PROGRAM SingleCarrierMode
VAR
	(*key Command*)
	btn_Power:BOOL;
	btn_PowerOn: BOOL;
	btn_PowerOff: BOOL;
	TopPositionNew:LREAL:=100;
	TopVelocityNew:LREAL:=1;
	btn_TopMove:BOOL;
	btn_TopStop:BOOL;
	BottomPositionNew:LREAL:=100;
	BottomVelocityNew:LREAL:=1;
	btn_BottomMove:BOOL;
	btn_BottomStop:BOOL;
	(*Var*)
	fb_ton1:TON;
	fb_ton2:TON;
	fb_ton3:TON;
	(*Status*)
	State:DINT;
	Busy:BOOL;
	TopBusy:BOOL;
	BottomBusy:BOOL;
	InitDone:BOOL;
	tm_state: DINT;
	ts_state: DINT;
	bm_state: DINT;
	bs_state: DINT;
	(*PowerOff*)
	d_state: DINT;
	(*¼ì²âµ½ÏÞÎ»£¬»Ö¸´Move×´Ì¬*)
	FTrig_ReachLS: F_TRIG;
	FTrig_btn_GapMove: F_TRIG;
END_VAR

TopPositionActual:=(Pos_LeftTopLin+Pos_RightTopLin)/2;
TopVelocityActual:=(Velo_LeftTopLin+Velo_RightTopLin)/2;
BottomPositionActual:=(Pos_LeftBottomLin+Pos_RightBOttomLin)/2;
BottomVelocityActual:=(Velo_LeftBottomLin+Velo_RightBOttomLin)/2;
(*********************************************************************btn_PowerOn************************************************************)
IF btn_Power AND st_Power=0 THEN
	btn_PowerOn:=TRUE;
	btn_Power:=FALSE;
END_IF
IF btn_Power AND st_Power=1 THEN
	btn_PowerOff:=TRUE;
	btn_Power:=FALSE;
END_IF
(*********************************************************************btn_PowerOn************************************************************)

IF btn_PowerOn THEN
	A_CoupleAxisAndPowerOn();
END_IF
(******************************************************ÉÏµç×´Ì¬£¬²»´¦ÓÚñîºÏ×´Ì¬£¬ESTOP***********************************************)
IF NOT btn_PowerOff THEN
	IF st_Power=1 AND st_Couple<>1THEN
		Error:=TRUE;
		ErrorID:=101;
		FB_PlcEmergencyStop();
		LED_Error:=TRUE;
	END_IF
END_IF
(*********************************************************************Monitor All Carrirt Position***********************************************)
A_MonitoringAllAxis();
(*********************************************************************A_PosDiffDetection***********************************************)
A_PosDiffDetection();
(*********************************************************************btn_TopMove*****************************************************************)
IF InitDone THEN
	IF btn_TopMove AND NOT bottomBusy THEN
		TopBusy:=TRUE;
		btn_BottomMove:=FALSE;
		CASE tm_state OF
			0:
				FB_Move.Mode:=2;						(*1£ºgapÄ£Ê½£»2£ºµ¥ÁºÄ£Ê½£¬3£ºtaperÄ£Ê½*)
				FB_Move.CoupleState:=st_Couple;			(*ñîºÏ×´Ì¬ÊäÈë*)
				FB_Move.PowerState:=st_Power;			(*µçÔ´×´Ì¬ÊäÈë*)
				FB_Move.TopMove:=TRUE;				(*Execute TRUE*)
				FB_Move.TopPosition:=TopPositionNew;		(*Î»ÖÃ*)
				FB_Move.TopVelocity:=TopVelocityNew;		(*ËÙ¶È*)
				FB_Move();								(*Æô¶¯FB*)
				IF TopPositionNew-TopPositionActual>0.001 THEN	(*ÔË¶¯·½ÏòÖ¸Ê¾*)
					TopMoveIndicator:=1;
				ELSIF TopPositionNew-TopPositionActual<0.001 THEN
					TopMoveIndicator:=-1;
				ELSE
					TopMoveIndicator:=0;
				END_IF
				tm_state:=1;
			1:
				FB_Move();
				LED_Run:=TRUE;
				IF NOT FB_Move.TopDone THEN			(*ÔË¶¯Î´Íê³É£¬Ñ­»·*)
					tm_state:=1;
				ELSE									(*ÔË¶¯Íê³É£¬ÏÂÒ»²½*)
					tm_state:=88;
				END_IF
			88:
				btn_TopMove:=FALSE;					(*×´Ì¬»Ö¸´*)
				LED_Run:=FALSE;
				tm_state:=0;
				TopBusy:=FALSE;
		END_CASE
	END_IF
END_IF

(*********************************************************************btn_BottomMove*****************************************************************)
IF InitDone THEN
	IF btn_BottomMove AND NOT TopBusy THEN
		btn_TopMove:=FALSE;
		BottomBusy:=TRUE;
		CASE bm_state OF
			0:
				FB_Move.Mode:=2;						(*1£ºgapÄ£Ê½£»2£ºµ¥ÁºÄ£Ê½£¬3£ºtaperÄ£Ê½*)
				FB_Move.CoupleState:=st_Couple;			(*ñîºÏ×´Ì¬ÊäÈë*)
				FB_Move.PowerState:=st_Power;			(*µçÔ´×´Ì¬ÊäÈë*)
				FB_Move.BottomMove:=TRUE;				(*Execute TRUE*)
				FB_Move.BottomPosition:=BottomPositionNew;		(*Î»ÖÃ*)
				FB_Move.BottomVelocity:=BottomVelocityNew;		(*ËÙ¶È*)
				FB_Move();								(*Æô¶¯FB*)
				IF BottomPositionNew-BottomPositionActual>0.001 THEN	(*ÔË¶¯·½ÏòÖ¸Ê¾*)
					BottomMoveIndicator:=1;
				ELSIF BottomPositionNew-BottomPositionActual<0.001 THEN
					BottomMoveIndicator:=-1;
				ELSE
					BottomMoveIndicator:=0;
				END_IF
				bm_state:=1;
			1:
				FB_Move();
				IF NOT FB_Move.BottomDone THEN			(*ÔË¶¯Î´Íê³É£¬Ñ­»·*)
					LED_Run:=TRUE;
					bm_state:=1;
				ELSE									(*ÔË¶¯Íê³É£¬ÏÂÒ»²½*)
					bm_state:=88;
				END_IF
			88:
				BottomBusy:=FALSE;
				btn_TopMove:=FALSE;
				btn_BottomMove:=FALSE;					(*×´Ì¬»Ö¸´*)
				bm_state:=0;
				LED_Run:=FALSE;
		END_CASE
	END_IF
END_IF
(*******************************************************************btn_TopStop********************************************************************)
IF btn_TopStop THEN
	LED_Run:=FALSE;
	TopMoveIndicator:=0;
	FB_Move.TopReset:=TRUE;								(*¸øÔË¶¯FB¸øÍ£Ö¹ÐÅºÅ£¬Ê¹FB_Move×´Ì¬»Ö¸´*)
	TopBusy:=FALSE;
	FB_Move();											(*Æô¶¯FB_Move*)
	btn_TopMove:=FALSE;									(*btn_GapMove:=FALSE*)
	tm_state:=0;											(*m_state:=0;*)
	CASE ts_state OF
			0:
				FB_Stop.Mode:=2;							(*1£ºgapÄ£Ê½£»2£ºµ¥ÁºÄ£Ê½£»3£ºtaperÄ£Ê½*)
				FB_Stop.CoupleState:=st_Couple;			(*ñîºÏ×´Ì¬ÊäÈë*)
				FB_Stop.PowerState:=st_Power;				(*µçÔ´×´Ì¬ÊäÈë*)
				FB_Stop.TopStop:=TRUE;					(*Execute TRUE*)
				FB_Stop();								(*Æô¶¯FB*)
				ts_state:=1;
			1:
				FB_Stop();
				IF NOT FB_Stop.TopDone THEN			(*Í£Ö¹Î´Íê³É£¬Ñ­»·*)
					ts_state:=1;
				ELSE									(*Í£Ö¹Íê³É£¬ÏÂÒ»²½*)
					ts_state:=88;
				END_IF
			88:
				btn_TopStop:=FALSE;						(*»Ö¸´×´Ì¬*)
				FB_Move.TopReset:=FALSE;					(*ÔËÐÐFB*)
				ts_state:=0;
		END_CASE
END_IF
(*******************************************************************btn_BottomStop********************************************************************)
IF btn_BottomStop  THEN
	LED_Run:=FALSE;
	BottomMoveIndicator:=0;
	FB_Move.BottomReset:=TRUE;								(*¸øÔË¶¯FB¸øÍ£Ö¹ÐÅºÅ£¬Ê¹FB_Move×´Ì¬»Ö¸´*)
	BottomBusy:=FALSE;
	FB_Move();											(*Æô¶¯FB_Move*)
	btn_BottomMove:=FALSE;									(*btn_GapMove:=FALSE*)
	bm_state:=0;											(*m_state:=0;*)
	CASE bs_state OF
			0:
				FB_Stop.Mode:=2;							(*1£ºgapÄ£Ê½£»2£ºµ¥ÁºÄ£Ê½£»3£ºtaperÄ£Ê½*)
				FB_Stop.CoupleState:=st_Couple;			(*ñîºÏ×´Ì¬ÊäÈë*)
				FB_Stop.PowerState:=st_Power;				(*µçÔ´×´Ì¬ÊäÈë*)
				FB_Stop.BottomStop:=TRUE;					(*Execute TRUE*)
				FB_Stop();								(*Æô¶¯FB*)
				bs_state:=1;
			1:
				FB_Stop();
				IF NOT FB_Stop.BottomDone THEN			(*Í£Ö¹Î´Íê³É£¬Ñ­»·*)
					bs_state:=1;
				ELSE									(*Í£Ö¹Íê³É£¬ÏÂÒ»²½*)
					bs_state:=88;
				END_IF
			88:
				btn_BottomStop:=FALSE;						(*»Ö¸´×´Ì¬*)
				FB_Move.BottomReset:=FALSE;					(*ÔËÐÐFB*)
				bs_state:=0;
		END_CASE
END_IF
(*********************************************************************btn_PowerOff************************************************************)
IF btn_PowerOff THEN
	A_DecoupleAndPowerOff();
END_IF
(*********************************************************************ÏÞÎ»Åö´¥×´Ì¬»Ö¸´************************************************************)
(*Èç¹û¼ì²âµ½ÏØÏÞÎ»¿ª¹ØÏÂ½µÑØ£¬»Ö¸´Move×´Ì¬*)
FTrig_ReachLS(CLK:=Unreach_LS_Top AND Unreach_LS_Bottom);
IF FTrig_ReachLS.Q THEN		(*FTrig_ReachLS.QÌ«¿ì£¬Ö»ÄÜÊ¹btn_TopStopÎªTRUE*)
	btn_TopStop:=TRUE;
	btn_BottomStop:=TRUE;
END_IF
IF btn_TopStop THEN			(*Òò´Ë£¬´Ë´¦Îªµ±Ö®Ç°btn_TopStopÎªTRUEÊ±£¬ÈËÎªÈÃbtn_BottomStopÎªTRUE*)
	btn_BottomStop:=TRUE;
END_IF
(*Èç¹û¼ì²âµ½TopÏÞÎ»¿ª¹ØFALSE£¬ÇÒÄ¿±êÎ»ÖÃ´óÓÚµ±Ç°Î»ÖÃÊ±£¬»òÕßÏà·´Ê±£¬»Ö¸´Move×´Ì¬*)
IF NOT Unreach_LS_Top AND TopPositionNew-TopPositionActual>0.0005 AND btn_TopMove THEN
	btn_TopStop:=TRUE;
END_IF
IF NOT Unreach_LS_Bottom AND TopPositionNew-TopPositionActual<0.0005 AND btn_TopMove THEN
	btn_TopStop:=TRUE;
END_IF
IF NOT Unreach_LS_Top AND BottomPositionNew-BottomPositionActual>0.0005 AND btn_BottomMove THEN
	btn_BottomStop:=TRUE;
END_IF
IF NOT Unreach_LS_Bottom AND BottomPositionNew-BottomPositionActual<0.0005 AND btn_BottomMove THEN
	btn_BottomStop:=TRUE;
END_IF

ACTION A_CoupleAxisAndPowerOn:
(****************************************************************
NAME:			A_SetAxisPositionAndCoupleAxisAndPowerOn
DATA:			2017.3.20
VERSION:		1.0.0
DESCRIPTION:	
				ÉÏµãÃüÁîºó£¬Ë³ÐòÖ´ÐÐ£º
				1.FB_SetAxisPosition
				2.FB_CoupleAxis
				3.FB_PowerOn
				·µ»ØÖ´ÐÐÊÇ·ñ³É¹¦
HISTORY:
				2017.3.20		NEW

***************************************************************)
fb_ton2(PT:=t#0.5s);
fb_ton3(PT:=t#0.5S);
CASE State OF
	0:	(*FB_Couple_Axis*)
		FB_CoupleAxis(Execute:=TRUE);
		fb_ton2.IN:=TRUE;
		State:=1;
	1:	(*wait*)
		FB_CoupleAxis();
		IF NOT FB_CoupleAxis.InGear THEN		(*FB_Couple_AxisÃ»ÓÐÖ´ÐÐÍê£¬wait£¬³¬Ê±FB Error*)
			IF NOT fb_ton1.Q THEN
				State:=1;
			ELSE
				ErrorID:=1;
				State:=99;
			END_IF
		ELSE
			State:=2;
		END_IF
	2:	(*FB_Power_On*)
		FB_Power(On:=TRUE);
		fb_ton3.IN:=TRUE;
		State:=3;
	3:	(*wait*)
		FB_power();
		IF NOT FB_power.OnStatus THEN		(*FB_Power_OnÃ»ÓÐÖ´ÐÐÍê£¬wait£¬³¬Ê±FB Error*)
			IF NOT fb_ton3.Q THEN
				State:=3;
			ELSE
				ErrorID:=2;
				State:=99;
			END_IF
		ELSE
			State:=88;
		END_IF
	88:	(*All Done*)
		btn_PowerOn:=FALSE;
		State:=0;
		Error:=FALSE;
		ErrorID:=0;
		Busy:=FALSE;
		InitDone:=TRUE;
		FB_CoupleAxis.Execute:=FALSE;
		FB_power.On:=FALSE;
		fb_ton1.IN:=FALSE;
		fb_ton2.IN:=FALSE;
		fb_ton3.IN:=FALSE;
	99:
		btn_PowerOn:=FALSE;
		State:=99;
		Error:=TRUE;
		Busy:=FALSE;
		InitDone:=FALSE;
		FB_CoupleAxis.Execute:=FALSE;
		FB_Power.On:=FALSE;
		fb_ton1.IN:=FALSE;
		fb_ton2.IN:=FALSE;
		fb_ton3.IN:=FALSE;
		LED_Error:=TRUE;
END_CASE
END_ACTION

ACTION A_DecoupleAndPowerOff:
FB_DecoupleAxis();
CASE d_state OF
		0:(*Decouple*)
			FB_DecoupleAxis.Execute:=TRUE;
			FB_DecoupleAxis();
			d_state:=1;
		1:
			IF NOT FB_DecoupleAxis.OutGear THEN
				d_state:=1;
			ELSE
				d_state:=2;
			END_IF
		2:(*PowerOff*)
			FB_Power(Off:=TRUE);
				d_state:=3;
		3:
			IF NOT FB_power.OffStatus THEN
				d_state:=3;
			ELSE
				d_state:=88;
			END_IF
		88:(*ResetAllState*)
			btn_PowerOn:=FALSE;
			btn_TopMove:=FALSE;
			btn_TopStop:=FALSE;
			btn_BottomMove:=FALSE;
			btn_BottomStop:=FALSE;
			fb_ton1.IN:=FALSE;
			fb_ton2.IN:=FALSE;
			fb_ton3.IN:=FALSE;
			State:=0;
			Busy:=FALSE;
			TopBusy:=FALSE;
			BottomBusy:=FALSE;
			InitDone:=FALSE;
			Error:=FALSE;
			ErrorID:=0;
			bm_state:=0;
			bs_state:=0;
			tm_state:=0;
			ts_state:=0;
			btn_PowerOff:=FALSE;
			d_state:=0;
			FB_DecoupleAxis.Execute:=FALSE;
			FB_DecoupleAxis.Reset:=TRUE;
			FB_DecoupleAxis();
			FB_CoupleAxis.Execute:=FALSE;
			FB_CoupleAxis.Reset:=TRUE;
			FB_CoupleAxis();
			LED_Error:=FALSE;
			LED_Run:=FALSE;
END_CASE
END_ACTION

ACTION A_MonitoringAllAxis:
(****************************************************************
NAME:			A_MonitoringAllAxis
DATA:			2017.3.20
VERSION:		1.0.0
DESCRIPTION:	
				Ã¿´ÎÑ­»·¾ùÖ´ÐÐÖáÎ»ÖÃºÍÖáÔË¶¯µÄ¼ì²é
				1.4ÖáÏà¶ÔÔË¶¯¼ì²é
				2.4Öá¹âÕ¤³ßÎ»ÖÃ¡¢ËÙ¶È¶Ô±È¼ì²é
				3.Ã¿Öá¹âÕ¤ºÍ±àÂëÆ÷Î»ÖÃ¶Ô±È¼ì²é
HISTORY:
				2017.3.20		NEW

***************************************************************)
(*************************************************************************************1.4ÖáÏà¶ÔÔË¶¯¼ì²é************************************************************************************)
(*1Öá¶¯£¬ÆäËüÈýÖá²»¶¯*)
IF  (LeftTopLin.Status.Moving AND NOT RightTopLin.Status.NotMoving AND NOT  LeftBottomLin.Status.NotMoving AND NOT RightBottomLin.Status.NotMoving)
	OR (NOT LeftTopLin.Status.NotMoving AND RightTopLin.Status.Moving AND NOT LeftBottomLin.Status.NotMoving AND NOT RightBottomLin.Status.NotMoving)
	OR (NOT LeftTopLin.Status.NotMoving AND NOT RightTopLin.Status.NotMoving AND LeftBottomLin.Status.Moving AND NOT  RightBottomLin.Status.NotMoving)
	OR (NOT LeftTopLin.Status.NotMoving AND NOT RightTopLin.Status.NotMoving AND NOT LeftBottomLin.Status.NotMoving AND RightBottomLin.Status.Moving) THEN
		btn_TopStop:=TRUE;
		btn_BottomStop:=TRUE;
		FB_PlcEmergencyStop();
		Error:=TRUE;
		ErrorID:=11;
		LED_Error:=TRUE;
(*2Öá¶¯£¬2Öá²»¶¯(µ¥ÁºÁ½Öá¶¯Õý³£)*)
ELSIF  (LeftTopLin.Status.Moving AND NOT RightTopLin.Status.Moving AND LeftBottomLin.Status.Moving AND NOT RightBottomLin.Status.Moving)
	OR  (NOT LeftTopLin.Status.Moving AND  RightTopLin.Status.Moving AND  NOT LeftBottomLin.Status.Moving AND  RightBottomLin.Status.Moving) THEN
		btn_TopStop:=TRUE;
		btn_BottomStop:=TRUE;
		FB_PlcEmergencyStop();
		Error:=TRUE;
		ErrorID:=12;
		LED_Error:=TRUE;
(*3Öá¶¯£¬1Öá²»¶¯*)
ELSIF  (NOT LeftTopLin.Status.NotMoving AND RightTopLin.Status.Moving AND LeftBottomLin.Status.Moving AND RightBottomLin.Status.Moving)
	OR  (LeftTopLin.Status.Moving AND NOT RightTopLin.Status.NotMoving AND LeftBottomLin.Status.Moving AND RightBottomLin.Status.Moving)
	OR  (LeftTopLin.Status.Moving AND RightTopLin.Status.Moving AND NOT  LeftBottomLin.Status.NotMoving AND RightBottomLin.Status.Moving)
	OR  (LeftTopLin.Status.Moving AND RightTopLin.Status.Moving AND LeftBottomLin.Status.Moving AND NOT RightBottomLin.Status.NotMoving) THEN
		btn_TopStop:=TRUE;
		btn_BottomStop:=TRUE;
		FB_PlcEmergencyStop();
		Error:=TRUE;
		ErrorID:=13;
		LED_Error:=TRUE;
END_IF
(*************************************************************************************2.4Öá¹âÕ¤³ßÎ»ÖÃ¡¢ËÙ¶È¶Ô±È¼ì²é**********************************************************************)
IF  st_Power<>0 THEN
(*Top Î»ÖÃºÍËÙ¶È±È¶Ô*)
		Diff_TopPos_actual:=Pos_leftTopLin-Pos_RightTopLin;
		Diff_TopVelo_actual:=Velo_leftTopLin-Velo_RightTopLin;
IF ABS(Pos_leftTopLin-Pos_RightTopLin)>Threshold_TopPos_SingleCarrier THEN
		btn_TopStop:=TRUE;
		btn_BottomStop:=TRUE;
		FB_PlcEmergencyStop();
		Error:=TRUE;
		ErrorID:=14;
		LED_Error:=TRUE;
ELSIF ABS(Velo_leftTopLin-Velo_RightTopLin)>Threshold_TopVelo_SingleCarrier  THEN
		(*btn_TopStop:=TRUE;
		btn_BottomStop:=TRUE;
		FB_PlcEmergencyStop();*)
		Error:=TRUE;
		ErrorID:=15;
(*Bottom Î»ÖÃºÍËÙ¶È±È¶Ô*)
ELSIF ABS(Pos_LeftBottomLin-Pos_RightBottomLin)>Threshold_BottomPos_SingleCarrier THEN
		btn_TopStop:=TRUE;
		btn_BottomStop:=TRUE;
		FB_PlcEmergencyStop();
		Error:=TRUE;
		ErrorID:=16;
		LED_Error:=TRUE;
ELSIF ABS(Velo_leftBottomLin-Velo_RightBottomLin)>Threshold_BottomVelo_SingleCarrier  THEN
		(*btn_TopStop:=TRUE;
		btn_BottomStop:=TRUE;
		FB_PlcEmergencyStop();*)
		Error:=TRUE;
		ErrorID:=17;
(*ÎÞLeftºÍRightËÙ¶ÈÎ»ÖÃµÄ¶Ô±È*)
END_IF
END_IF
(*********************************************************************************3.Ã¿Öá¹âÕ¤ºÍ±àÂëÆ÷Î»ÖÃ¶Ô±È¼ì²é**********************************************************************)
END_ACTION

ACTION A_PosDiffDetection:
IF ABS(PosDiff_LeftTopLin_actual-PosDiff_RightTopLin_actual)>0.2 THEN
	ErrorID:=51;
	Error:=TRUE;
	btn_TopStop:=TRUE;
	btn_BottomStop:=TRUE;
	FB_PlcEmergencyStop();
	LED_Error:=TRUE;
ELSIF ABS(PosDiff_LeftBottomLin_actual-PosDiff_RightBottomLin_actual)>0.2 THEN
	ErrorID:=53;
	Error:=TRUE;
	btn_TopStop:=TRUE;
	btn_BottomStop:=TRUE;
	FB_PlcEmergencyStop();
	LED_Error:=TRUE;
END_IF
END_ACTION

END_PROGRAM

(* stored: Version 1.1.0.1, ProductVersion 3.1.4024.6
   POU SingleCarrierMode: Id {932b8545-d89d-46a8-8a71-7d229764fd43}, SpecialFunc None
   Action A_CoupleAxisAndPowerOn: Id {0ef71d57-a8c3-4101-ab11-36cd3c0eca26}
   Action A_DecoupleAndPowerOff: Id {4f0ea523-0b13-4621-8f4d-b9142410fd56}
   Action A_MonitoringAllAxis: Id {eb43239b-219b-4196-a91d-cc3c414c514e}
   Action A_PosDiffDetection: Id {e36b8bee-016d-4e0e-8a51-c5aff2c5ba67} *)
